FUNCTION_BLOCK TEST_SH (* Test bit shift functions *)
  (* Standard: 61499-1 *)
  (* Version 0.1, 2007-11-11, JHC, Holobloc Inc, Deleted import. *)
  (* Version 0.0, 2006-09-06, JHC, Holobloc Inc *)
  (* Compiler header: package fb.rt.test; *)
  (* Compiler classdef: SimpleFB *)
  (* Compiler Java Sun JDK 1.6.0 *)
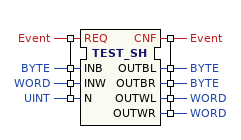
  EVENT_INPUT
    REQ WITH INB, INW, N; (* Normal Execution Request *)
  END_EVENT
  EVENT_OUTPUT
    CNF WITH OUTBL, OUTBR, OUTWL, OUTWR; (* Execution Confirmation *)
  END_EVENT
  VAR_INPUT
    INB : BYTE;
    INW : WORD;
    N : UINT;
  END_VAR
  VAR_OUTPUT
    OUTBL : BYTE;
    OUTBR : BYTE;
    OUTWL : WORD;
    OUTWR : WORD;
  END_VAR
  ALGORITHM REQ IN FBD: (* Normally executed algorithm *)
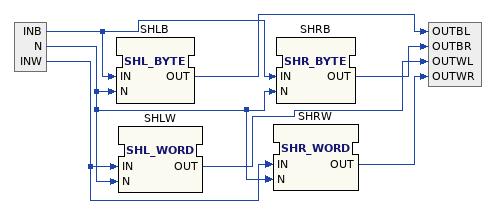
    FBS
      SHLB : SHL_BYTE;
      SHRB : SHR_BYTE;
      SHLW : SHL_WORD;
      SHRW : SHR_WORD;
    END_FBS
    DATA_CONNECTIONS
      INB TO SHLB.IN;
      N TO SHLB.N;
      SHLB.OUT TO OUTBL;
      INB TO SHRB.IN;
      N TO SHRB.N;
      SHRB.OUT TO OUTBR;
      INW TO SHLW.IN;
      N TO SHLW.N;
      SHLW.OUT TO OUTWL;
      INW TO SHRW.IN;
      N TO SHRW.N;
      SHRW.OUT TO OUTWR;
    END_CONNECTIONS
  END_ALGORITHM
END_FUNCTION_BLOCK
